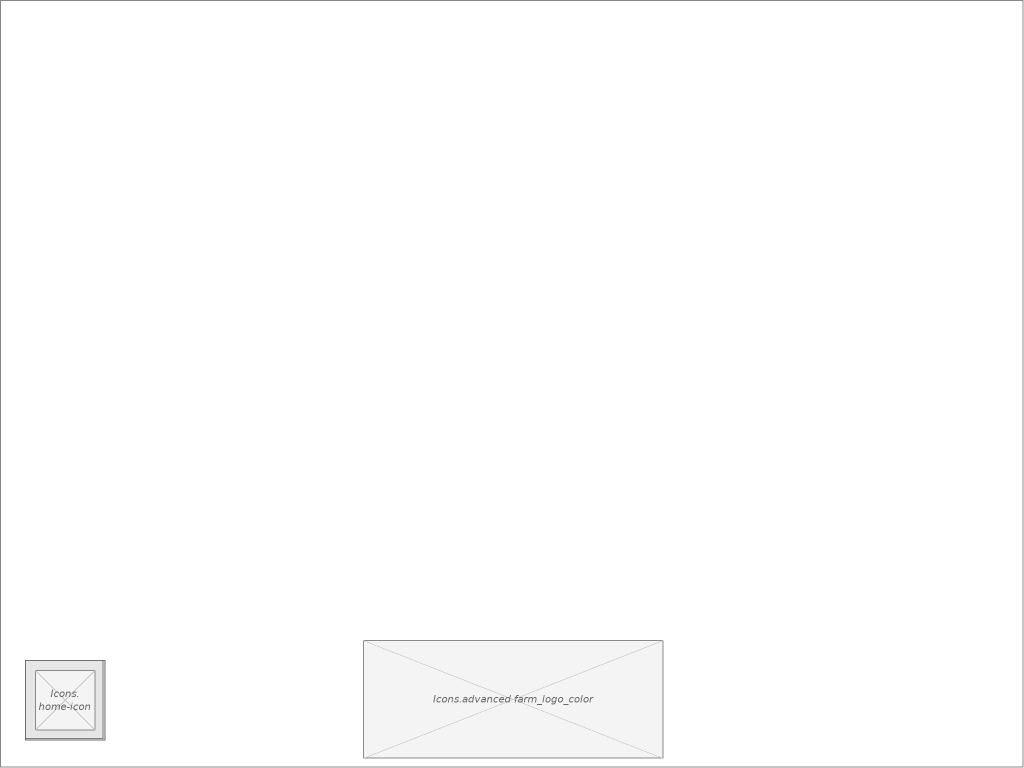
VISUALIZATION Stats_Screen  // 1024x768
    Image (363,640 300x118), image: Icons.advanced farm_logo_color
    Group (25,660 80x80)
        OnMouseClick: change screen: Home_Screen
        Button (0,0 80x80)
        Image (10,10 60x60), image: Icons.home-icon
END_VISUALIZATION

(* stored: Version 1.1.0.1, ProductVersion 3.1.4024.15
   Visu Stats_Screen: Id {31767a78-5a9a-4c7d-a9ea-d000761d1951} *)
